// TIA Portal V17 export
// export: Created 2026-04-13T11:12:05.0249871Z, ExportSetting WithDefaults, DisplayName Totally Integrated Automation Portal, DisplayVersion V17 Update 4, DisplayName TIA Portal Openness, DisplayVersion V17 Update 4, DisplayName TIA Portal Version Control Interface, DisplayVersion V17, DisplayName SINAMICS Startdrive Advanced, DisplayVersion V17, DisplayName SINAMICS Startdrive G130, G150, S120, S150, SINAMICS MV, S210, DisplayVersion V17, DisplayName SINAMICS Startdrive G110M, G120, G120C, G120D, G120P, G115D, DisplayVersion V17, DisplayName STEP 7 Professional, DisplayVersion V17 Update 4, DisplayName STEP 7 Safety, DisplayVersion V17, DisplayName WinCC Professional, DisplayVersion V17 Update 4
DATA_BLOCK "CIP_CUS"   // DB6
{ S7_Optimized_Access := 'FALSE' }
VERSION : 0.1
// stored: AutoNumber true, DBAccessibleFromOPCUA true, DBAccessibleFromWebserver true, IsOnlyStoredInLoadMemory false, IsWriteProtectedInAS false
   VAR
      RCV : Struct
         QXT心跳信号 : Bool;
         QCIP启动 : Bool;
         QCS纯水洗 : Bool;
         QJS碱水洗 : Bool;
         QRJ溶剂洗 : Bool;
         QYK压空阀 : Bool;
         QRS热水洗 : Bool;
         QSJ水进程泵 : Bool;
         QRJ溶剂进程泵 : Bool;
         QXY泄压请求 : Bool;
         QQS缺水状态 : Bool;
         QQX清洗模式状态 : Int;
         QJX碱洗温度 : Real;
         QJS碱水液位 : Real;
         QCS纯水温度 : Real;
         QCS纯水液位 : Real;
         QRJ溶剂温度 : Real;
         QRJ溶剂液位 : Real;
         QJC碱纯压力 : Real;
         QCS溶剂压力 : Real;
      END_STRUCT;
      Send : Struct
         MXT心跳信号 : Bool;
         MBM北面喷雾 : Bool;
         MCS纯水模块洗 : Bool;
         MJS碱水模块洗 : Bool;
         MRJ溶剂模块洗 : Bool;
         MRS热水模块洗 : Bool;
         MCS纯水洗 : Bool;
         MJX碱洗 : Bool;
         MRJ溶剂洗 : Bool;
         MYK压空阀 : Bool;
         MRS热水洗 : Bool;
         MSJ水进程泵 : Bool;
         MRJ溶剂进程泵 : Bool;
         MGS供水泵 : Bool;
         MXY泄压阀 : Bool;
         MQX清洗模式 : Int;
         MPW喷雾模式 : Real;
         MJX碱洗温度设定 : Real := 80.0;
         MPS排水时间 : Real;
      END_STRUCT;
   END_VAR
BEGIN
END_DATA_BLOCK
